// TIA Portal V16 export
// export: Created 2023-03-29T11:04:45.1270606Z, ExportSetting WithDefaults, DisplayName Totally Integrated Automation Portal, DisplayVersion V16 Update 6, DisplayName TIA Portal Version Control Interface, DisplayVersion V16 Update 2, DisplayName TIA Portal Openness, DisplayVersion V16 Update 6, DisplayName STEP 7 Professional, DisplayVersion V16 Update 6, DisplayName STEP 7 Safety, DisplayVersion V16, DisplayName WinCC Advanced, DisplayVersion V16 Update 6
FUNCTION "Sterownik_P1P2P3P4" : Void   // FC3, LAD
{ S7_Optimized_Access := 'TRUE' }
AUTHOR : RTecmer
VERSION : 0.1
// Sterowaniepompownią
// Funkcja zarządza sygnałem załączającym styczniki (sieć), (Falownik) danego napędu
// Sterowanie kompresorami
// Algorytm przewiduje sterowanie nadrzędne w trybie automatycznym przez sterownik master "OMROM". Sterowanie w trybie Manual z systemu SCADA odbywa się przez sterownik SLAVE "S7-1200" . Sterownik S7-100 reguluje sygnałem zadawania Hz w oparciu o regulator PID. Sygnał ten podawany jest na wejście analogowe sterownika Master. Praca sterownika S7-1200 Slave ogranicza się do generowania sygnału Hz, wystawianiu sygnału Automat, sygnału Dodatkowy kompresor 1, sygnału Dodatkowy kompresor 2. Komunikacji z systemem SCADA.
// stored: AutoNumber true, IsIECCheckEnabled false, SetENOAutomatically false, UDAEnableTagReadback false
BEGIN

REGION Network 1: Drive P1 / P1 Driver
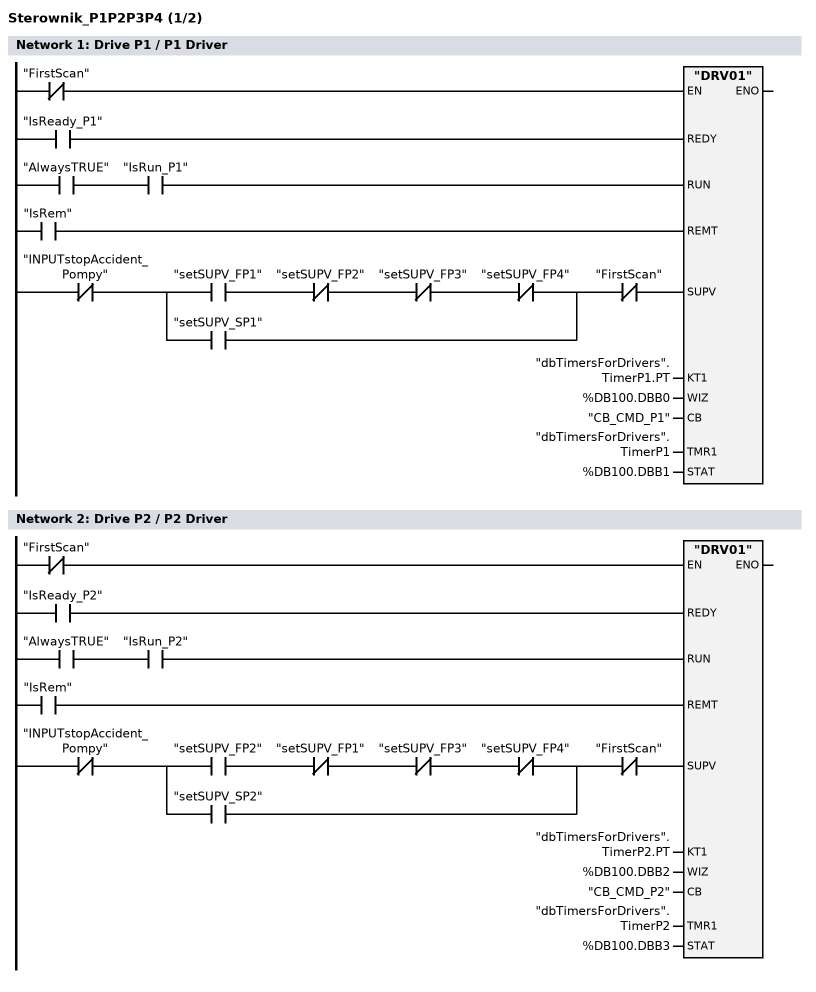
   RUNG wire#powerrail
      I_Contact( "FirstScan" )
      "DRV01"(REDY := wire#w1, RUN := wire#w2, REMT := wire#w3, SUPV := wire#w6, KT1 := "dbTimersForDrivers".TimerP1.PT, WIZ := %DB100.DBB0, CB := "CB_CMD_P1", TMR1 := "dbTimersForDrivers".TimerP1, STAT := %DB100.DBB1)
   END_RUNG
   RUNG wire#powerrail
      Contact( "IsReady_P1" )
   END_RUNG wire#w1
   RUNG wire#powerrail
      Contact( "AlwaysTRUE" )
      Contact( "IsRun_P1" )
   END_RUNG wire#w2
   RUNG wire#powerrail
      Contact( "IsRem" )
   END_RUNG wire#w3
   RUNG wire#powerrail
      I_Contact( "INPUTstopAccident_Pompy" )
      wire#w4
      Contact( "setSUPV_FP1" )
      I_Contact( "setSUPV_FP2" )
      I_Contact( "setSUPV_FP3" )
      I_Contact( "setSUPV_FP4" )
      wire#w5
      I_Contact( "FirstScan" )
   END_RUNG wire#w6
   RUNG wire#w4
      Contact( "setSUPV_SP1" )
   END_RUNG wire#w5
   // the same network as SCL:
   IF NOT "FirstScan" THEN
       "DRV01"(REDY := "IsReady_P1",
               RUN := "AlwaysTRUE" AND "IsRun_P1",
               REMT := "IsRem",
               SUPV := NOT "INPUTstopAccident_Pompy" AND (("setSUPV_FP1" AND NOT "setSUPV_FP2" AND NOT "setSUPV_FP3" AND NOT "setSUPV_FP4") OR "setSUPV_SP1") AND NOT "FirstScan",
               KT1 := "dbTimersForDrivers".TimerP1.PT,
               WIZ := %DB100.DBB0,
               CB := "CB_CMD_P1",
               TMR1 := "dbTimersForDrivers".TimerP1,
               STAT := %DB100.DBB1);
   END_IF;
END_REGION

REGION Network 2: Drive P2 / P2 Driver
   RUNG wire#powerrail
      I_Contact( "FirstScan" )
      "DRV01"(REDY := wire#w1, RUN := wire#w2, REMT := wire#w3, SUPV := wire#w6, KT1 := "dbTimersForDrivers".TimerP2.PT, WIZ := %DB100.DBB2, CB := "CB_CMD_P2", TMR1 := "dbTimersForDrivers".TimerP2, STAT := %DB100.DBB3)
   END_RUNG
   RUNG wire#powerrail
      Contact( "IsReady_P2" )
   END_RUNG wire#w1
   RUNG wire#powerrail
      Contact( "AlwaysTRUE" )
      Contact( "IsRun_P2" )
   END_RUNG wire#w2
   RUNG wire#powerrail
      Contact( "IsRem" )
   END_RUNG wire#w3
   RUNG wire#powerrail
      I_Contact( "INPUTstopAccident_Pompy" )
      wire#w4
      Contact( "setSUPV_FP2" )
      I_Contact( "setSUPV_FP1" )
      I_Contact( "setSUPV_FP3" )
      I_Contact( "setSUPV_FP4" )
      wire#w5
      I_Contact( "FirstScan" )
   END_RUNG wire#w6
   RUNG wire#w4
      Contact( "setSUPV_SP2" )
   END_RUNG wire#w5
   // the same network as SCL:
   IF NOT "FirstScan" THEN
       "DRV01"(REDY := "IsReady_P2",
               RUN := "AlwaysTRUE" AND "IsRun_P2",
               REMT := "IsRem",
               SUPV := NOT "INPUTstopAccident_Pompy" AND (("setSUPV_FP2" AND NOT "setSUPV_FP1" AND NOT "setSUPV_FP3" AND NOT "setSUPV_FP4") OR "setSUPV_SP2") AND NOT "FirstScan",
               KT1 := "dbTimersForDrivers".TimerP2.PT,
               WIZ := %DB100.DBB2,
               CB := "CB_CMD_P2",
               TMR1 := "dbTimersForDrivers".TimerP2,
               STAT := %DB100.DBB3);
   END_IF;
END_REGION

REGION Network 3: Drive P3 / P3 Driver
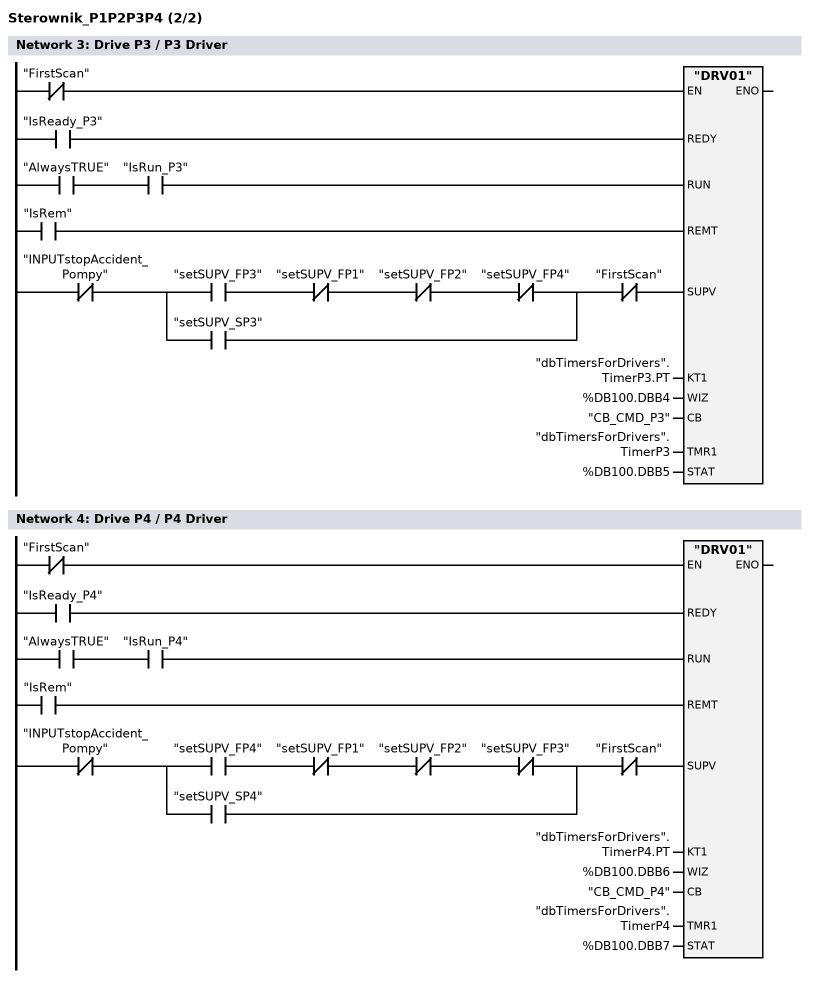
   RUNG wire#powerrail
      I_Contact( "FirstScan" )
      "DRV01"(REDY := wire#w1, RUN := wire#w2, REMT := wire#w3, SUPV := wire#w6, KT1 := "dbTimersForDrivers".TimerP3.PT, WIZ := %DB100.DBB4, CB := "CB_CMD_P3", TMR1 := "dbTimersForDrivers".TimerP3, STAT := %DB100.DBB5)
   END_RUNG
   RUNG wire#powerrail
      Contact( "IsReady_P3" )
   END_RUNG wire#w1
   RUNG wire#powerrail
      Contact( "AlwaysTRUE" )
      Contact( "IsRun_P3" )
   END_RUNG wire#w2
   RUNG wire#powerrail
      Contact( "IsRem" )
   END_RUNG wire#w3
   RUNG wire#powerrail
      I_Contact( "INPUTstopAccident_Pompy" )
      wire#w4
      Contact( "setSUPV_FP3" )
      I_Contact( "setSUPV_FP1" )
      I_Contact( "setSUPV_FP2" )
      I_Contact( "setSUPV_FP4" )
      wire#w5
      I_Contact( "FirstScan" )
   END_RUNG wire#w6
   RUNG wire#w4
      Contact( "setSUPV_SP3" )
   END_RUNG wire#w5
   // the same network as SCL:
   IF NOT "FirstScan" THEN
       "DRV01"(REDY := "IsReady_P3",
               RUN := "AlwaysTRUE" AND "IsRun_P3",
               REMT := "IsRem",
               SUPV := NOT "INPUTstopAccident_Pompy" AND (("setSUPV_FP3" AND NOT "setSUPV_FP1" AND NOT "setSUPV_FP2" AND NOT "setSUPV_FP4") OR "setSUPV_SP3") AND NOT "FirstScan",
               KT1 := "dbTimersForDrivers".TimerP3.PT,
               WIZ := %DB100.DBB4,
               CB := "CB_CMD_P3",
               TMR1 := "dbTimersForDrivers".TimerP3,
               STAT := %DB100.DBB5);
   END_IF;
END_REGION

REGION Network 4: Drive P4 / P4 Driver
   RUNG wire#powerrail
      I_Contact( "FirstScan" )
      "DRV01"(REDY := wire#w1, RUN := wire#w2, REMT := wire#w3, SUPV := wire#w6, KT1 := "dbTimersForDrivers".TimerP4.PT, WIZ := %DB100.DBB6, CB := "CB_CMD_P4", TMR1 := "dbTimersForDrivers".TimerP4, STAT := %DB100.DBB7)
   END_RUNG
   RUNG wire#powerrail
      Contact( "IsReady_P4" )
   END_RUNG wire#w1
   RUNG wire#powerrail
      Contact( "AlwaysTRUE" )
      Contact( "IsRun_P4" )
   END_RUNG wire#w2
   RUNG wire#powerrail
      Contact( "IsRem" )
   END_RUNG wire#w3
   RUNG wire#powerrail
      I_Contact( "INPUTstopAccident_Pompy" )
      wire#w4
      Contact( "setSUPV_FP4" )
      I_Contact( "setSUPV_FP1" )
      I_Contact( "setSUPV_FP2" )
      I_Contact( "setSUPV_FP3" )
      wire#w5
      I_Contact( "FirstScan" )
   END_RUNG wire#w6
   RUNG wire#w4
      Contact( "setSUPV_SP4" )
   END_RUNG wire#w5
   // the same network as SCL:
   IF NOT "FirstScan" THEN
       "DRV01"(REDY := "IsReady_P4",
               RUN := "AlwaysTRUE" AND "IsRun_P4",
               REMT := "IsRem",
               SUPV := NOT "INPUTstopAccident_Pompy" AND (("setSUPV_FP4" AND NOT "setSUPV_FP1" AND NOT "setSUPV_FP2" AND NOT "setSUPV_FP3") OR "setSUPV_SP4") AND NOT "FirstScan",
               KT1 := "dbTimersForDrivers".TimerP4.PT,
               WIZ := %DB100.DBB6,
               CB := "CB_CMD_P4",
               TMR1 := "dbTimersForDrivers".TimerP4,
               STAT := %DB100.DBB7);
   END_IF;
END_REGION
END_FUNCTION
